{attribute 'qualified_only'}
TYPE eTcaCarrierLayout :
(
	undefined := 0,
	Layout1,
	Layout2,
	Layout3,
	Layout4,
	Layout5,
	Bulk
);
END_TYPE

(* stored: Version 1.1.0.1
   DUT eTcaCarrierLayout: Id {79b55d49-ef51-4dd5-9342-bb36d3007c7b} *)
